// Block: A0301_PERS

DATA_BLOCK A0301_PERS
VERSION : 0.1
   NON_RETAIN
   VAR
      Par : Struct
         Maint_FreeMove : Bool;
         CaseA_PLen_Lim : Real;
         CaseA_StopperSensor : USInt;
         CaseB_PLen_Lim : Real;
         CaseB_StopperSensor : USInt;
         CaseC_PLen_Lim : Real;
         CaseC_StopperSensor : USInt;
         CaseD_PLen_Lim : Real;
         CaseD_StopperSensor : USInt;
         DlySensorsON : Time;
         DlySensorsOFF : Time;
         TolReachNextStopper : Real;
         TolReachAllSensorsON : Real;
      END_STRUCT;
      Par_Mng : Struct
         DlySensorsON : Time;
         DlySensorsOFF : Time;
         TRK : Struct
            BTrk_MoveP4Exit : Time;
            BTrk_MoveToP5 : Time;
         END_STRUCT;
      END_STRUCT;
      Data_Mng : Struct
         LastCounter_PartMove_P2toP4 : LReal;
         LastCounter_PartMove_P1toP2 : LReal;
         LastCounter_PartMove_P1toP3 : LReal;
      END_STRUCT;
      FC_Sensor : Struct
         "Case" : Int;
      END_STRUCT;
      SensTime : Struct
         P1 : Struct
            Sens_Ing : Struct
               DelayOn : Time;
            END_STRUCT;
            Sens_Out : Struct
               DelayOff : Time;
            END_STRUCT;
         END_STRUCT;
         P2 : Struct
            Sens_Ing : Struct
               DelayOn : Time;
            END_STRUCT;
            Sens_Out : Struct
               DelayOff : Time;
            END_STRUCT;
         END_STRUCT;
         P3 : Struct
            Sens_Ing : Struct
               DelayOn : Time;
            END_STRUCT;
            Sens_Out : Struct
               DelayOff : Time;
            END_STRUCT;
         END_STRUCT;
         P4 : Struct
            Sens_Ing : Struct
               DelayOn : Time;
            END_STRUCT;
            Sens_Out : Struct
               DelayOff : Time;
            END_STRUCT;
         END_STRUCT;
      END_STRUCT;
   END_VAR

BEGIN
   // No initialization required
END_DATA_BLOCK
